FUNCTION_BLOCK fTemp
VAR_INPUT
	iAnalog:INT;
END_VAR
VAR_OUTPUT	
	rValue:REAL;
END_VAR

VAR
	A: INT;
END_VAR

(*-------------------------------------------------------------------------------------------------------*)
A:= A+1;
(*Conversion UF a temperatura ºC*)
rValue :=INT_TO_REAL(iAnalog)/10.0;

END_FUNCTION_BLOCK

(* stored: Version 1.1.0.1, ProductVersion 3.1.4024.10
   POU fTemp: Id {5849953f-bdb4-4f35-9702-6e3af3710252}, SpecialFunc None *)
